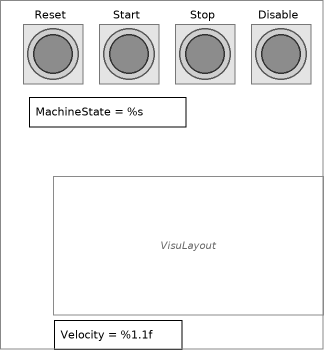
VISUALIZATION Visualization  // 324x350
    Rectangle (29,97 157x30), "MachineState = %s", text variable: MAIN.MachineState
    PushSwitch (23,24 60x60), variable: MAIN.HmiReset, behaviour: TAP, style: Switch-PushSwitch-Gray
    Label (18,5 65x20), "Reset"
    PushSwitch (99,24 60x60), variable: MAIN.HmiRun, behaviour: TAP, style: Switch-PushSwitch-Gray
    Label (94,5 65x20), "Start"
    PushSwitch (175,24 60x60), variable: MAIN.HmiStop, behaviour: TAP, style: Switch-PushSwitch-Gray
    Label (170,5 65x20), "Stop"
    Frame (53,176 271x139)
        shows VisuLayout()
    Rectangle (54,320 128x30), "Velocity = %1.1f", text variable: GVL.MoverVelo
        OnMouseClick: write the text variable via Default, min 5, max 2000
    PushSwitch (251,24 60x60), variable: MAIN.HmiDisable, behaviour: TAP, style: Switch-PushSwitch-Gray
    Label (246,5 65x20), "Disable"
END_VISUALIZATION

(* stored: Version 1.1.0.1, ProductVersion 3.1.4024.12
   Visu Visualization: Id {b7dac3b3-97e1-45dc-9b36-68910ba6e024} *)
